TYPE TYP_FAULHABER_SC_HW :
STRUCT
	In : TYP_FAULHABER_SC_HW_IN;
	Out : TYP_FAULHABER_SC_HW_OUT;
END_STRUCT
END_TYPE

(* stored: Version 1.1.0.1, ProductVersion 3.1.4024.12
   DUT TYP_FAULHABER_SC_HW: Id {7928c25c-96a3-4613-85f9-4ab838f5c38c} *)
